// TIA Portal V17 export
FUNCTION "Motor_Control" : Void   // FC, LAD
{ S7_Optimized_Access := 'TRUE' }
VERSION : 0.1
// stored: AutoNumber true, IsIECCheckEnabled false, SetENOAutomatically false
BEGIN

REGION Network 1
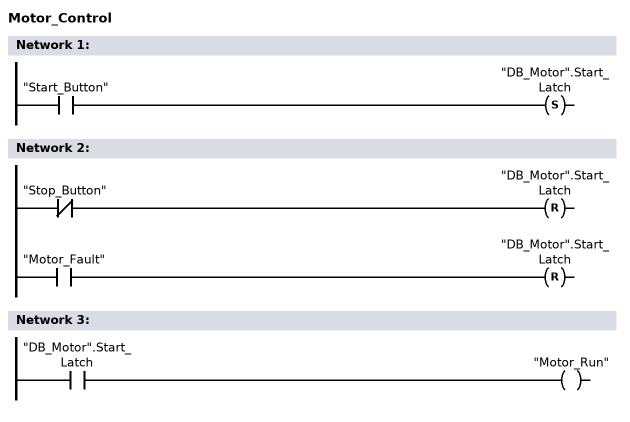
   RUNG wire#powerrail
      Contact( "Start_Button" )
      S_Coil( "DB_Motor".Start_Latch )
   END_RUNG
   // the same network as SCL:
   IF "Start_Button" THEN "DB_Motor".Start_Latch := TRUE; END_IF;
END_REGION

REGION Network 2
   RUNG wire#powerrail
      I_Contact( "Stop_Button" )
      R_Coil( "DB_Motor".Start_Latch )
   END_RUNG
   RUNG wire#powerrail
      Contact( "Motor_Fault" )
      R_Coil( "DB_Motor".Start_Latch )
   END_RUNG
   // the same network as SCL:
   IF NOT "Stop_Button" THEN "DB_Motor".Start_Latch := FALSE; END_IF;
   IF "Motor_Fault" THEN "DB_Motor".Start_Latch := FALSE; END_IF;
END_REGION

REGION Network 3
   RUNG wire#powerrail
      Contact( "DB_Motor".Start_Latch )
      Coil( "Motor_Run" )
   END_RUNG
   // the same network as SCL:
   "Motor_Run" := "DB_Motor".Start_Latch;
END_REGION
END_FUNCTION
